FUNCTION "SM_StateFirstCall" : Bool
{ S7_Optimized_Access := 'FALSE' }
VERSION : 0.1
   VAR_IN_OUT
      inst : "typeSM";
   END_VAR


BEGIN
	#SM_StateFirstCall := #inst.stateChanged AND (#inst.stateTime > T#0ms);
END_FUNCTION

